FUNCTION_BLOCK SkillGoToRight (* Basic Function Block Type *)
  (* Standard: 61499-2 *)
  (* Version 0.0, 2/16/2024, midxav, Template *)
  PACKAGE Main;
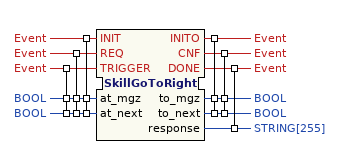
  EVENT_INPUT
    INIT WITH at_mgz, at_next; (* Initialization Request *)
    REQ WITH at_mgz, at_next; (* Normal Execution Request *)
    TRIGGER WITH at_mgz, at_next;
  END_EVENT
  EVENT_OUTPUT
    INITO WITH to_mgz, to_next; (* Initialization Confirm *)
    CNF WITH to_mgz, to_next; (* Execution Confirmation *)
    DONE WITH response;
  END_EVENT
  VAR_INPUT
    at_mgz : BOOL;
    at_next : BOOL;
  END_VAR
  VAR_OUTPUT
    to_mgz : BOOL;
    to_next : BOOL;
    response : STRING[255];
  END_VAR
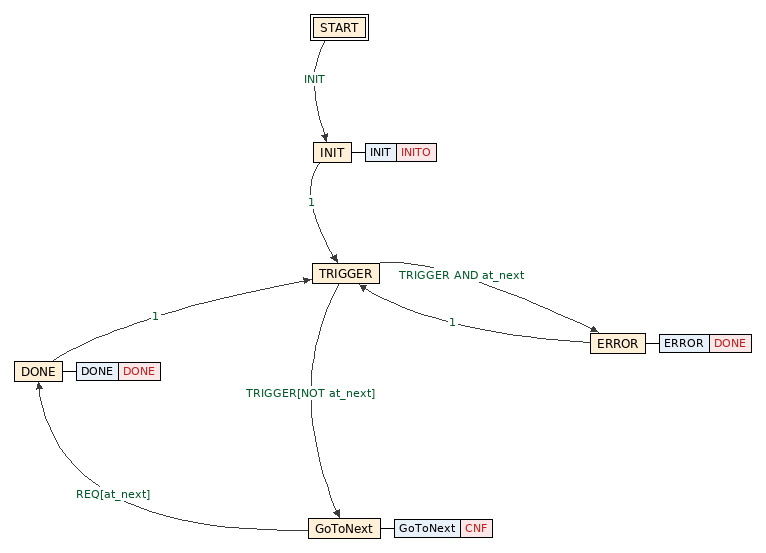
  EC_STATES
    START; (* Initial State *)
    INIT : INIT -> INITO; (* Initialization *)
    GoToNext : GoToNext -> CNF;
    DONE : DONE -> DONE;
    TRIGGER;
    ERROR : ERROR -> DONE;
  END_STATES
  EC_TRANSITIONS
    START TO INIT := INIT;
    TRIGGER TO GoToNext := TRIGGER[NOT at_next];
    GoToNext TO DONE := REQ[at_next];
    DONE TO TRIGGER := 1;
    INIT TO TRIGGER := 1;
    TRIGGER TO ERROR := TRIGGER AND at_next;
    ERROR TO TRIGGER := 1;
  END_TRANSITIONS
  ALGORITHM INIT IN ST: (* Initialization algorithm *)
to_mgz :=FALSE;
to_next :=FALSE;
response:='INITIALISED';
  END_ALGORITHM
  ALGORITHM GoToMag IN ST:
to_mgz := TRUE;
to_next := FALSE;
response:='MOVED TO STORAGE';
  END_ALGORITHM
  ALGORITHM GoToNext IN ST:
to_mgz := FALSE;
to_next := TRUE;
response:='MOVING TO RIGHT';
  END_ALGORITHM
  ALGORITHM DONE IN ST:
response:='MOVED TO RIGHT';
  END_ALGORITHM
  ALGORITHM ERROR IN ST:
response:='ALREADY AT RIGHT SIDE';
TRIGGER:=FALSE;
  END_ALGORITHM
END_FUNCTION_BLOCK
